// TIA Portal V18 export
VAR_GLOBAL   // PLC tag table "Output"
   "Left Driver On/Off output" AT %Q0.0 : Bool;
   "Left Driver Reversing output" AT %Q0.1 : Bool;
   "Left Driver Fault output" AT %Q0.2 : Bool;
   "Left Driver DI4 STO output" AT %Q0.3 : Bool;
   "Left Driver DI5 STO output" AT %Q0.4 : Bool;
   "Right Driver On/Off output" AT %Q0.5 : Bool;
   "Right Driver Reversing output" AT %Q0.6 : Bool;
   "Right Driver Fault output" AT %Q0.7 : Bool;
   "Right Driver DI4 STO output" AT %Q1.0 : Bool;
   "Right Driver DI5 STO output" AT %Q1.1 : Bool;
   "Cab Driver On/Off output" AT %Q2.0 : Bool;
   "Cab Driver Reversing output" AT %Q2.1 : Bool;
   "Cab Driver Fault Reset output" AT %Q2.2 : Bool;
   "Cab Driver DI4 STO output" AT %Q2.3 : Bool;
   "Cab Driver DI5 STO output" AT %Q2.4 : Bool;
   "Left & Right Warning Lights output" AT %Q2.5 : Bool;   // R3 -
   "Mania Lights output" AT %Q2.7 : Bool;   // R5 -
   "Motor Brake Left output" AT %Q3.4 : Bool;   // R10 -
   "Motor Brake Right output" AT %Q3.5 : Bool;   // R11 -
   "Cabin Motor Brake output" AT %Q3.6 : Bool;   // R13 -
   "Cab Warning Light & Buzzer output" AT %Q3.7 : Bool;   // R4 -
   "Valve Up output" AT %Q4.0 : Bool;   // R14 -
   "Valve Em Down output" AT %Q4.1 : Bool;   // R15 -
   "Valve Down output" AT %Q4.2 : Bool;   // R16 -
   "Valve V4 Columns" AT %Q4.3 : Bool;   // R17 -
   "Valve  V5 Columns" AT %Q4.4 : Bool;   // R18 -
   "MC - Main Contactor output" AT %Q5.0 : Bool;
   "Hydraulic output" AT %Q5.1 : Bool;   // C1 - MC-105, MC-106, MC-107, MC-108, Cable No:200, MKS2
   "Tunnel Lighting A" AT %Q5.3 : Bool;   // C3 (A
   "Tunnel Lighting B" AT %Q5.4 : Bool;   // C4 (B
   "Tunnel Lighting C" AT %Q5.5 : Bool;   // C5 (C
   "Hose power output" AT %Q7.1 : Bool;   // C2 -
   "SafetyShoe Activated output" AT %Q7.2 : Bool;   // R24 -
   "PBB On output" AT %Q7.3 : Bool;   // R20 -
   "Safety Edge Reset output" AT %Q7.4 : Bool;   // DBX in Relay Reset
   "Fire Detector output" AT %Q8.0 : Bool;   // R25 -
   "SafetyShoe Power output" AT %Q8.2 : Bool;   // R51 -
   "PCA Active OUT output" AT %Q8.3 : Bool;
   "GPU1 Active OUT output" AT %Q8.4 : Bool;
   "GPU2 Active OUT output" AT %Q8.5 : Bool;
   "AutoLeveller Fault output" AT %Q8.6 : Bool;   // R23 -
   "PBB Autoleveler ON output" AT %Q9.0 : Bool;
   "Autoleveller On output" AT %Q9.1 : Bool;   // R22 -
   "PBB HOME output" AT %Q9.2 : Bool;
   "SafetyEdge Red Light output" AT %Q9.3 : Bool;   // R1 - MC-256 MC-257 MC-258, Cable No:204, F11
   "Bumper Red Light iptal output" AT %Q9.4 : Bool;   // R2 -
   "Ext Lighting output" AT %Q3.0 : Bool;   // C5 -
   "Tunnel Lights UPS output" AT %Q9.6 : Bool;   // C4 -
   "PBB Error/Fault/Alarm output" AT %Q9.7 : Bool;   // R21 -
   "AutoLeveller FW output" AT %Q10.2 : Bool;   // C9 -
   "AutoLeveller BW output" AT %Q10.3 : Bool;   // C10
   "Left Canopy FW output" AT %Q10.6 : Bool;   // C13
   "Left Canopy BW output" AT %Q10.7 : Bool;   // C14
   "Right Canopy FW output" AT %Q11.0 : Bool;   // C15
   "Right Canopy BW output" AT %Q11.1 : Bool;   // C16
   "Cab Floor FW output" AT %Q11.2 : Bool;   // C50
   "Cab Floor BW output" AT %Q11.3 : Bool;   // C51
   "CP - Buzzer output" AT %Q12.0 : Bool;
   "CP - Alarm Red Light output" AT %Q12.1 : Bool;
   "CP - PBB Start Green Light output" AT %Q12.2 : Bool;
   "CP - Reset Red Light output" AT %Q12.3 : Bool;
   "CP - Button Int Lighting Light output" AT %Q12.4 : Bool;
   "CP - Button Ext Lighting Light output" AT %Q12.5 : Bool;
   "CP - Button Em Stop Light output" AT %Q12.7 : Bool;
   "Cab Warning Light output" AT %Q2.6 : Bool;
   "Ext Lighting Projector output" AT %Q3.1 : Bool;
   "CP - Button Ext Lighting Projector output" AT %Q12.6 : Bool;
   "Air Conditions Trigger" AT %Q4.5 : Bool;   // R19 (
END_VAR
